FUNCTION_BLOCK Test_FB_Counter_SetsQ_Output EXTENDS T_UnitTestBase
VAR
    Counter : CTU;
END_VAR

// Setup..
Counter(
	CU:= FALSE, 
	RESET:= TRUE, 
	PV:= 1, 
	Q=> , 
	CV=> );

// Test... 
Counter(
	CU:= TRUE, 
	RESET:= FALSE, 
	PV:= , 
	Q=> , 
	CV=> );
// Verify...   
Assertion.AssertEquals_BOOL(
    Expected:= TRUE, 
    Actual:= Counter.Q, 
    VariableName:= 'Counter.Q');   

// Done...   
TestFinished();

END_FUNCTION_BLOCK

(* stored: Version 1.1.0.1, ProductVersion 3.1.4024.6
   POU Test_FB_Counter_SetsQ_Output: Id {c08e92b5-5880-4083-ba7d-60b1332265cf}, SpecialFunc None *)
